	                    #sFB_Conveyor570(iUDT_ConveyorConfiguration := #iUDT_Configuration."570".Conveyor,
	                                     idi_PECEoSDistance := #iUDT_Configuration."570".PEC_Eos.Distance,
	                                     idi_PECBoSDistance := 0,
	                                     ii_ExternalSpeed := 0,
	                                     ix_SafetyOk := #ix_SafetyOk,
	                                     ix_24vOk := #ix_24vOk,
	                                     ix_400vOk := #ix_400vOk,
	                                     ix_HardwareOk := #iUDT_HardwareOk."570",
	                                     ix_PECEoS := #iqUDT_WorkstationStatus."570".PEC_EoS.PEC,
	                                     ix_PECBoS := TRUE,
	                                     ix_ExternalRequestHold := #sx_RightExternalRequestHold570,
	                                     qUDT_HMIStatus => #iqUDT_WorkstationStatus."570".Conveyor,
	                                     qUDT_Status => #iqUDT_WorkstationCommonStatus."570",
	                                     iqUDT_EquipmentControl := #iqUDT_EquipmentControl,
	                                     iqUDT_ConveyorCommand := #iqUDT_WorkstationCommands."570".Conveyor,
	                                     iqUDT_ConveyorInterface := #sUDT_Interface570,
	                                     iqUDT_HandShakeUp := #sUDT_Handshake560,
	                                     iqUDT_HandShake := #sUDT_Handshake570,
	                                     iqUDT_Statistics := #iqUDT_WorkstationStatistics."570".Conveyor);
	                END_REGION

	                REGION MCO

	                    #sFB_MCOConveyLinxAixController570(iUDT_AixConfig := #iUDT_Configuration."570".MCO_M01,
	                                                       iv_AixInputsModule := #iUDT_MotorInput570,
	                                                       ix_24vOk := #ix_24vOk,
	                                                       ix_SimulationModeActive := "DB_Memory".Simulation,
	                                                       ii_MotorPositionId := 1,
	                                                       qUDT_HMIStatus => #iqUDT_WorkstationStatus."570".MCO_M01,
	                                                       iqv_AixOutputsModule := #iqUDT_MotorOutput570,
	                                                       iqUDT_ConveyorInterface := #sUDT_Interface570,
	                                                       iqUDT_MCOStatistics := #iqUDT_WorkstationStatistics."570".MCO_M01);
	                END_REGION
	            END_REGION

	            REGION 580

	                REGION Displacement

	                    #sFB_Displacement580(#sUDT_Interface580);

	                END_REGION

	                REGION Tracking

	                    #sFB_Tracking580(iUDT_ConveyorCommonConfiguration := #iUDT_Configuration."580".Conveyor.Common,
	                                     iqa_TrackingData := #sa_TrackingArray580,
	                                     iqUDT_ConveyorInterface := #sUDT_Interface580,
	                                     iqUDT_HandshakeUp := #sUDT_Handshake570,
	                                     iqUDT_Handshake := #sUDT_Handshake580);
	                END_REGION

	                REGION EOS

	                    #sFB_PECUpdate580(iUDT_PECUpdateConfiguration := #iUDT_Configuration."580".PEC_Eos,
	                                      iUDT_ConveyorCommonConfiguration := #iUDT_Configuration."580".Conveyor.Common,
	                                      ix_PEC := NOT #iUDT_MotorInput570.AllSensorPortInputs.RightSensor,
	                                      ix_TeachingMode := FALSE,
	                                      qUDT_Status => #iqUDT_WorkstationStatus."580".PEC_EoS,
	                                      qi_GINwrite => #ti_dummy,
	                                      qx_PECFiltered => #tx_dummy,
	                                      iqa_TrackingData := #sa_TrackingArray580,
	                                      iqUDT_ConveyorInterface := #sUDT_Interface580,
	                                      iqUDT_UnknownGINRange := #iqUDT_UnknownGINRange,
	                                      iqUDT_FifoHeader := "DB_FIFOLostGIN".Header,
	                                      iqa_FifoData := "DB_FIFOLostGIN".Data,
	                                      iqUDT_Statistics := #iqUDT_WorkstationStatistics."580".PEC_EoS);

	                END_REGION

	                REGION Conveyor

	                    #sUDT_Handshake580.RTR := #sx_RightIndexing AND
	                    ((#iqUDT_WorkstationStatus."590".PEC_EoS.PEC AND #sUDT_Interface590.ActualSpeed <> 0) OR #iqUDT_WorkstationStatus."580".PEC_EoS.PEC);

	                    #sFB_Conveyor580(iUDT_ConveyorConfiguration := #iUDT_Configuration."580".Conveyor,
	                                     idi_PECEoSDistance := #iUDT_Configuration."580".PEC_Eos.Distance,
	                                     idi_PECBoSDistance := 0,
	                                     ii_ExternalSpeed := 0,
	                                     ix_SafetyOk := #ix_SafetyOk,
	                                     ix_24vOk := #ix_24vOk,
	                                     ix_400vOk := #ix_400vOk,
	                                     ix_HardwareOk := #iUDT_HardwareOk."580",
	                                     ix_PECEoS := #iqUDT_WorkstationStatus."580".PEC_EoS.PEC,
	                                     ix_PECBoS := TRUE,
	                                     ix_ReverseDirection := FALSE,
	                                     ix_ExternalRequestDieBack := FALSE,
	                                     ix_ExternalRequestHold := #sx_RightExternalRequestHold580,
	                                     ix_ResetEnergySave := FALSE,
	                                     qUDT_HMIStatus => #iqUDT_WorkstationStatus."580".Conveyor,
	                                     qUDT_Status => #iqUDT_WorkstationCommonStatus."580",
	                                     iqUDT_EquipmentControl := #iqUDT_EquipmentControl,
	                                     iqUDT_ConveyorCommand := #iqUDT_WorkstationCommands."580".Conveyor,
	                                     iqUDT_ConveyorInterface := #sUDT_Interface580,
	                                     iqUDT_HandShakeUp := #sUDT_Handshake570,
	                                     iqUDT_HandShake := #sUDT_Handshake580,
	                                     iqUDT_Statistics := #iqUDT_WorkstationStatistics."580".Conveyor);
	                END_REGION

	                REGION MCO

	                    #sFB_MCOConveyLinxAixController580(iUDT_AixConfig := #iUDT_Configuration."580".MCO_M01,
	                                                       iv_AixInputsModule := #iUDT_MotorInput570,
	                                                       ix_24vOk := #ix_24vOk,
	                                                       ix_SimulationModeActive := "DB_Memory".Simulation,
	                                                       ii_MotorPositionId := 2,
	                                                       qUDT_HMIStatus => #iqUDT_WorkstationStatus."580".MCO_M01,
	                                                       iqv_AixOutputsModule := #iqUDT_MotorOutput570,
	                                                       iqUDT_ConveyorInterface := #sUDT_Interface580,
	                                                       iqUDT_MCOStatistics := #iqUDT_WorkstationStatistics."580".MCO_M01);
	                END_REGION

	            END_REGION

	            REGION 590

	                REGION Displacement

	                    #sFB_Displacement590(#sUDT_Interface590);

	                END_REGION

	                REGION Tracking

	                    #sFB_Tracking590(iUDT_ConveyorCommonConfiguration := #iUDT_Configuration."590".Conveyor.Common,
	                                     iqa_TrackingData := #sa_TrackingArray590,
	                                     iqUDT_ConveyorInterface := #sUDT_Interface590,
	                                     iqUDT_HandshakeUp := #sUDT_Handshake580,
	                                     iqUDT_Handshake := #sUDT_Handshake590);
	                END_REGION

	                REGION EOS

	                    #sFB_PECUpdate590(iUDT_PECUpdateConfiguration := #iUDT_Configuration."590".PEC_Eos,
	                                      iUDT_ConveyorCommonConfiguration := #iUDT_Configuration."590".Conveyor.Common,
	                                      ix_PEC := NOT #iUDT_MotorInput590.AllSensorPortInputs.LeftSensor,
	                                      ix_TeachingMode := FALSE,
	                                      qUDT_Status => #iqUDT_WorkstationStatus."590".PEC_EoS,
	                                      qi_GINwrite => #ti_dummy,
	                                      qx_PECFiltered => #tx_dummy,
	                                      iqa_TrackingData := #sa_TrackingArray590,
	                                      iqUDT_ConveyorInterface := #sUDT_Interface590,
	                                      iqUDT_UnknownGINRange := #iqUDT_UnknownGINRange,
	                                      iqUDT_FifoHeader := "DB_FIFOLostGIN".Header,
	                                      iqa_FifoData := "DB_FIFOLostGIN".Data,
	                                      iqUDT_Statistics := #iqUDT_WorkstationStatistics."590".PEC_EoS);

	                END_REGION

	                REGION Conveyor

	                    #sUDT_Handshake590.RTR := (#sx_RightIndexing AND #iqUDT_WorkstationStatus."590".PEC_EoS.PEC)
	                    OR (#sx_RightPushOutActiveStation1 AND #iqUDT_WorkstationStatus."610".PEC_EoS.PEC AND #sUDT_Interface611.ActualSpeed <> 0);

	                    #sFB_Conveyor590(iUDT_ConveyorConfiguration := #iUDT_Configuration."590".Conveyor,
	                                     idi_PECEoSDistance := #iUDT_Configuration."590".PEC_Eos.Distance,
	                                     idi_PECBoSDistance := 0,
	                                     ii_ExternalSpeed := 0,
	                                     ix_SafetyOk := #ix_SafetyOk,
	                                     ix_24vOk := #ix_24vOk,
	                                     ix_400vOk := #ix_400vOk,
	                                     ix_HardwareOk := #iUDT_HardwareOk."590",
	                                     ix_PECEoS := #iqUDT_WorkstationStatus."590".PEC_EoS.PEC,
	                                     ix_PECBoS := TRUE,
	                                     ix_ReverseDirection := FALSE,
	                                     ix_ExternalRequestDieBack := FALSE,
	                                     ix_ExternalRequestHold := #sx_RightExternalRequestHold590,
	                                     ix_ResetEnergySave := FALSE,
	                                     qUDT_HMIStatus => #iqUDT_WorkstationStatus."590".Conveyor,
	                                     qUDT_Status => #iqUDT_WorkstationCommonStatus."590",
	                                     iqUDT_EquipmentControl := #iqUDT_EquipmentControl,
	                                     iqUDT_ConveyorCommand := #iqUDT_WorkstationCommands."590".Conveyor,
	                                     iqUDT_ConveyorInterface := #sUDT_Interface590,
	                                     iqUDT_HandShakeUp := #sUDT_Handshake580,
	                                     iqUDT_HandShake := #sUDT_Handshake590,
	                                     iqUDT_Statistics := #iqUDT_WorkstationStatistics."590".Conveyor);
	                END_REGION

	                REGION MCO

	                    #sFB_MCOConveyLinxAixController590(iUDT_AixConfig := #iUDT_Configuration."590".MCO_M01,
	                                                       iv_AixInputsModule := #iUDT_MotorInput590,
	                                                       ix_24vOk := #ix_24vOk,
	                                                       ix_SimulationModeActive := "DB_Memory".Simulation,
	                                                       ii_MotorPositionId := 1,
	                                                       qUDT_HMIStatus => #iqUDT_WorkstationStatus."590".MCO_M01,
	                                                       iqv_AixOutputsModule := #iqUDT_MotorOutput590,
	                                                       iqUDT_ConveyorInterface := #sUDT_Interface590,
	                                                       iqUDT_MCOStatistics := #iqUDT_WorkstationStatistics."590".MCO_M01);
	                END_REGION
	            END_REGION

	            REGION 610

	                REGION Displacement

	                    #sFB_Displacement610(#sUDT_Interface610);

	                END_REGION

	                REGION MCO

	                    #sFB_MCOConveyLinxAixController610(iUDT_AixConfig := #iUDT_Configuration."610".MCO_M01,
	                                                       iv_AixInputsModule := #iUDT_MotorInput610,
	                                                       ix_24vOk := #ix_24vOk,
	                                                       ix_SimulationModeActive := "DB_Memory".Simulation,
	                                                       ii_MotorPositionId := 1,
	                                                       qUDT_HMIStatus => #iqUDT_WorkstationStatus."610".MCO_M01,
	                                                       iqv_AixOutputsModule := #iqUDT_MotorOutput610,
	                                                       iqUDT_ConveyorInterface := #sUDT_Interface610,
	                                                       iqUDT_MCOStatistics := #iqUDT_WorkstationStatistics."610".MCO_M01);
	                END_REGION
	            END_REGION

	            REGION 611

	                REGION Displacement

	                    #sFB_Displacement611(#sUDT_Interface611);

	                END_REGION

	                REGION RAT

	                    #sFB_RightAngledTransfer611(iUDT_Configuration := #iUDT_Configuration."611".RightAngledTransfer,
	                                                iUDT_LowerConveyorConfiguration := #iUDT_Configuration."610".Conveyor,
	                                                iUDT_UpperConveyorConfiguration := #iUDT_Configuration."611".Conveyor,
	                                                iUDT_PECConfiguration := #iUDT_Configuration."610".PEC_EoS,
	                                                ii_DestinationA := 0,
	                                                ii_DestinationB := 0,
	                                                ii_DestinationC := 0,
	                                                ii_DestinationD := 2,
	                                                ix_HardwareOk := #iUDT_HardwareOk."610",
	                                                ix_400vOk := #ix_400vOk,
	                                                ix_24vOk := #ix_24vOk,
	                                                ix_SafetyOk := #ix_SafetyOk,
	                                                ix_AirPressureOk := #ix_AirPressureOk,
	                                                ix_SectionIsDown := #ix_SectionIsDown611,
	                                                ix_SectionIsUp := #ix_SectionIsUp611,
	                                                ix_ConveyorAAuto := false,
	                                                ix_ConveyorBAuto := false,
	                                                ix_ConveyorCAuto := FALSE,
	                                                ix_ConveyorDAuto := #iqUDT_WorkstationCommonStatus."590".AutoON,
	                                                ix_PEC := #iUDT_MotorInput610.AllSensorPortInputs.LeftSensor,
	                                                ix_ExternalReceiveRequestA := FALSE,
	                                                ix_ExternalReceiveRequestB := FALSE,
	                                                ix_ExternalReceiveRequestC := FALSE,
	                                                ix_ExternalReceiveRequestD := #sx_RightPushOutActiveStation1,
	                                                ix_PECInfeedD := #iqUDT_WorkstationStatus."590".PEC_EoS.PEC,
	                                                qUDT_HMIRATStatus => #iqUDT_WorkstationStatus."611".RightAngledTransfer,
	                                                qUDT_HMIConveyorStatus => #iqUDT_WorkstationStatus."610".Conveyor,
	                                                qUDT_HMIPECStatus => #iqUDT_WorkstationStatus."610".PEC_EoS,
	                                                qUDT_RATStatus => #iqUDT_WorkstationCommonStatus."611",
	                                                qUDT_ConveyorStatus => #iqUDT_WorkstationCommonStatus."610",
	                                                qx_PopupControl => #qx_PopupControl611,
	                                                qx_ExternalSendRequestA => #tx_dummy,
	                                                qx_ExternalSendRequestB => #tx_dummy,
	                                                qx_ExternalSendRequestC => #tx_dummy,
	                                                qx_ExternalSendRequestD => #tx_dummy,
	                                                iqUDT_EquipmentControl := #iqUDT_EquipmentControl,
	                                                iqUDT_RATCommand := #iqUDT_WorkstationCommands."611".RightAngledTransfer,
	                                                iqUDT_ConveyorCommand := #iqUDT_WorkstationCommands."610".Conveyor,
	                                                iqUDT_RATStatistics := #iqUDT_WorkstationStatistics."611".RightAngledTransfer,
	                                                iqUDT_ConveyorStatistics := #iqUDT_WorkstationStatistics."610".Conveyor,
	                                                iqUDT_PECStatistics := #iqUDT_WorkstationStatistics."610".PEC_EoS,
	                                                iqUDT_HandShakeConveyorA := #tUDT_DummyConveyorHandshake,
	                                                iqUDT_HandShakeConveyorB := #sUDT_Handshake610,
	                                                iqUDT_HandShakeConveyorC := #sUDT_Handshake590,
	                                                iqUDT_HandShakeConveyorD := #tUDT_DummyConveyorHandshake,
	                                                iqUDT_LowerConveyorInterface := #sUDT_Interface610,
	                                                iqUDT_UpperConveyorInterface := #sUDT_Interface611,
	                                                iqUDT_RATPositioning := #iqUDT_RATPositioning610,
	                                                iqUDT_BladeStopEoSInterface := #tUDT_DummyBladeStop,
	                                                iqUDT_BladeStopBoSInterface := #tUDT_DummyBladeStop);

	                END_REGION

	                REGION MCO

	                    #sFB_MCOConveyLinxAixController611(iUDT_AixConfig := #iUDT_Configuration."611".MCO_M01,
	                                                       iv_AixInputsModule := #iUDT_MotorInput610,
	                                                       ii_PositionSetpoint := #iqUDT_RATPositioning610.Upper.EndPosition,
	                                                       ix_24vOk := #ix_24vOk,
	                                                       ix_SimulationModeActive := "DB_Memory".Simulation,
	                                                       ii_MotorPositionId := 2,
	                                                       ix_StartPositioning := #iqUDT_RATPositioning610.Upper.Start,
	                                                       ix_ResetPosition := #iqUDT_RATPositioning610.Upper.ResetPosition,
	                                                       qUDT_HMIStatus => #iqUDT_WorkstationStatus."611".MCO_M01,
	                                                       qx_Positioned => #iqUDT_RATPositioning610.Upper.Done,
	                                                       iqv_AixOutputsModule := #iqUDT_MotorOutput610,
	                                                       iqUDT_ConveyorInterface := #sUDT_Interface611,
	                                                       iqUDT_MCOStatistics := #iqUDT_WorkstationStatistics."611".MCO_M01);
	                END_REGION

	            END_REGION

	            REGION 620

	                REGION Displacement

	                    #sFB_Displacement620(#sUDT_Interface620);

	                END_REGION

	                REGION MCO

	                    #sFB_MCOConveyLinxAixController620(iUDT_AixConfig := #iUDT_Configuration."620".MCO_M01,
	                                                       iv_AixInputsModule := #iUDT_MotorInput620,
	                                                       ii_PositionSetpoint := #iqUDT_RATPositioning620.Lower.EndPosition,
	                                                       ix_24vOk := #ix_24vOk,
	                                                       ix_SimulationModeActive := "DB_Memory".Simulation,
	                                                       ii_MotorPositionId := 1,
	                                                       ix_StartPositioning := #iqUDT_RATPositioning620.Lower.Start,
	                                                       ix_ResetPosition := #iqUDT_RATPositioning620.Lower.ResetPosition,
	                                                       qUDT_HMIStatus => #iqUDT_WorkstationStatus."620".MCO_M01,
	                                                       qx_Positioned => #iqUDT_RATPositioning620.Lower.Done,
	                                                       iqv_AixOutputsModule := #iqUDT_MotorOutput620,
	                                                       iqUDT_ConveyorInterface := #sUDT_Interface620,
	                                                       iqUDT_MCOStatistics := #iqUDT_WorkstationStatistics."620".MCO_M01);
	                END_REGION
	            END_REGION

	            REGION 621

	                REGION Displacement

	                    #sFB_Displacement621(#sUDT_Interface621);

	                END_REGION

	                REGION RAT

	                    #sFB_RightAngledTransfer621(iUDT_Configuration := #iUDT_Configuration."621".RightAngledTransfer,
	                                                iUDT_LowerConveyorConfiguration := #iUDT_Configuration."620".Conveyor,
	                                                iUDT_UpperConveyorConfiguration := #iUDT_Configuration."621".Conveyor,
	                                                iUDT_PECConfiguration := #iUDT_Configuration."620".PEC_EoS,
	                                                ii_DestinationA := 2,
	                                                ii_DestinationB := 0,
	                                                ii_DestinationC := 0,
	                                                ii_DestinationD := 2,
	                                                ix_HardwareOk := #iUDT_HardwareOk."620",
	                                                ix_400vOk := #ix_400vOk,
	                                                ix_24vOk := #ix_24vOk,
	                                                ix_SafetyOk := #ix_SafetyOk,
	                                                ix_AirPressureOk := #ix_AirPressureOk,
	                                                ix_SectionIsDown := #ix_SectionIsDown621,
	                                                ix_SectionIsUp := #ix_SectionIsUp621,
	                                                ix_ConveyorAAuto := #iqUDT_WorkstationCommonStatus."610".AutoON,
	                                                ix_ConveyorBAuto := false,
	                                                ix_ConveyorCAuto := false,
	                                                ix_ConveyorDAuto := #iqUDT_WorkstationCommonStatus."750".AutoON,
	                                                ix_PEC := #iUDT_MotorInput620.AllSensorPortInputs.LeftSensor,
	                                                ix_ExternalReceiveRequestA := NOT #iqUDT_WorkstationStatus."610".PEC_EoS.PEC,
	                                                ix_ExternalReceiveRequestB := FALSE,
	                                                ix_ExternalReceiveRequestC := FALSE,
	                                                ix_ExternalReceiveRequestD := NOT #iqUDT_WorkstationStatus."750".PEC_EoS.PEC,
	                                                ix_PECInfeedA := #iqUDT_WorkstationStatus."610".PEC_EoS.PEC,
	                                                ix_PECInfeedD := #iqUDT_WorkstationStatus."750".PEC_EoS.PEC,
	                                                qUDT_HMIRATStatus => #iqUDT_WorkstationStatus."621".RightAngledTransfer,
	                                                qUDT_HMIConveyorStatus => #iqUDT_WorkstationStatus."620".Conveyor,
	                                                qUDT_HMIPECStatus => #iqUDT_WorkstationStatus."620".PEC_EoS,
	                                                qUDT_RATStatus => #iqUDT_WorkstationCommonStatus."621",
	                                                qUDT_ConveyorStatus => #iqUDT_WorkstationCommonStatus."620",
	                                                qx_PopupControl => #qx_PopupControl621,
	                                                qx_ExternalSendRequestA => #tx_dummy,
	                                                qx_ExternalSendRequestB => #tx_dummy,
	                                                qx_ExternalSendRequestC => #tx_dummy,
	                                                qx_ExternalSendRequestD => #tx_dummy,
	                                                iqUDT_EquipmentControl := #iqUDT_EquipmentControl,
	                                                iqUDT_RATCommand := #iqUDT_WorkstationCommands."621".RightAngledTransfer,
	                                                iqUDT_ConveyorCommand := #iqUDT_WorkstationCommands."620".Conveyor,
	                                                iqUDT_RATStatistics := #iqUDT_WorkstationStatistics."621".RightAngledTransfer,
	                                                iqUDT_ConveyorStatistics := #iqUDT_WorkstationStatistics."620".Conveyor,
	                                                iqUDT_PECStatistics := #iqUDT_WorkstationStatistics."620".PEC_EoS,
	                                                iqUDT_HandShakeConveyorA := #sUDT_Handshake610,
	                                                iqUDT_HandShakeConveyorB := #iqUDT_HandshakeDownstream620,
	                                                iqUDT_HandShakeConveyorC := #tUDT_DummyConveyorHandshake,
	                                                iqUDT_HandShakeConveyorD := #sUDT_Handshake750,
	                                                iqUDT_LowerConveyorInterface := #sUDT_Interface620,
	                                                iqUDT_UpperConveyorInterface := #sUDT_Interface621,
	                                                iqUDT_RATPositioning := #iqUDT_RATPositioning620,
	                                                iqUDT_BladeStopEoSInterface := #tUDT_DummyBladeStop,
	                                                iqUDT_BladeStopBoSInterface := #tUDT_DummyBladeStop);

	                END_REGION

	                REGION MCO

	                    #sFB_MCOConveyLinxAixController621(iUDT_AixConfig := #iUDT_Configuration."621".MCO_M01,
	                                                       iv_AixInputsModule := #iUDT_MotorInput620,
	                                                       ii_PositionSetpoint := #iqUDT_RATPositioning620.Upper.EndPosition,
	                                                       ix_24vOk := #ix_24vOk,
	                                                       ix_SimulationModeActive := "DB_Memory".Simulation,
	                                                       ii_MotorPositionId := 2,
	                                                       ix_StartPositioning := #iqUDT_RATPositioning620.Upper.Start,
	                                                       ix_ResetPosition := #iqUDT_RATPositioning620.Upper.ResetPosition,
	                                                       qUDT_HMIStatus => #iqUDT_WorkstationStatus."621".MCO_M01,
	                                                       qx_Positioned => #iqUDT_RATPositioning620.Upper.Done,
	                                                       iqv_AixOutputsModule := #iqUDT_MotorOutput620,
	                                                       iqUDT_ConveyorInterface := #sUDT_Interface621,
	                                                       iqUDT_MCOStatistics := #iqUDT_WorkstationStatistics."621".MCO_M01);
	                END_REGION

	            END_REGION

	            REGION 710

	                REGION Displacement

	                    #sFB_Displacement710(#sUDT_Interface710);

	                END_REGION

	                REGION EOS
	                    #sFB_PEC710(ix_PEC := NOT #iUDT_MotorInput710.AllSensorPortInputs.LeftSensor,
	                                iUDT_PECConfiguration := #iUDT_Configuration."710".PEC_Eos,
	                                qx_PECFiltered => #tx_dummy,
	                                qUDT_HMIStatus => #iqUDT_WorkstationStatus."710".PEC_EoS,
	                                iqUDT_ConveyorInterface := #sUDT_Interface710,
	                                iqUDT_PECStatistics := #iqUDT_WorkstationStatistics."710".PEC_EoS);

	                END_REGION

	                REGION Conveyor

	                    #sFB_Conveyor710(iUDT_ConveyorConfiguration := #iUDT_Configuration."710".Conveyor,
	                                     idi_PECEoSDistance := #iUDT_Configuration."710".PEC_Eos.Distance,
	                                     idi_PECBoSDistance := 0,
	                                     ii_ExternalSpeed := 0,
	                                     ix_SafetyOk := #ix_SafetyOk,
	                                     ix_24vOk := #ix_24vOk,
	                                     ix_400vOk := #ix_400vOk,
	                                     ix_HardwareOk := #iUDT_HardwareOk."710",
	                                     ix_PECEoS := #iqUDT_WorkstationStatus."710".PEC_EoS.PEC,
	                                     ix_PECBoS := TRUE,
	                                     ix_ReverseDirection := FALSE,
	                                     ix_ExternalRequestDieBack := FALSE,
	                                     ix_ExternalRequestHold := #sx_RightExternalRequestHold710,
	                                     ix_ResetEnergySave := FALSE,
	                                     qUDT_HMIStatus => #iqUDT_WorkstationStatus."710".Conveyor,
	                                     qUDT_Status => #iqUDT_WorkstationCommonStatus."710",
	                                     iqUDT_EquipmentControl := #iqUDT_EquipmentControl,
	                                     iqUDT_ConveyorCommand := #iqUDT_WorkstationCommands."710".Conveyor,
	                                     iqUDT_ConveyorInterface := #sUDT_Interface710,
	                                     iqUDT_HandShakeUp := #tUDT_DummyConveyorHandshake,
	                                     iqUDT_HandShake := #sUDT_Handshake710,
	                                     iqUDT_Statistics := #iqUDT_WorkstationStatistics."710".Conveyor);
	                END_REGION

	                REGION MCO

	                    #sFB_MCOConveyLinxAixController710(iUDT_AixConfig := #iUDT_Configuration."710".MCO_M01,
	                                                       iv_AixInputsModule := #iUDT_MotorInput710,
	                                                       ix_24vOk := #ix_24vOk,
	                                                       ix_SimulationModeActive := "DB_Memory".Simulation,
	                                                       ii_MotorPositionId := 1,
	                                                       qUDT_HMIStatus => #iqUDT_WorkstationStatus."710".MCO_M01,
	                                                       iqv_AixOutputsModule := #iqUDT_MotorOutput710,
	                                                       iqUDT_ConveyorInterface := #sUDT_Interface710,
	                                                       iqUDT_MCOStatistics := #iqUDT_WorkstationStatistics."710".MCO_M01);
	                END_REGION

	            END_REGION

	            REGION 720

	                REGION Displacement

	                    #sFB_Displacement720(#sUDT_Interface720);

	                END_REGION

	                REGION EOS
	                    #sFB_PEC720(ix_PEC := NOT #iUDT_MotorInput710.AllSensorPortInputs.RightSensor,
	                                iUDT_PECConfiguration := #iUDT_Configuration."720".PEC_Eos,
	                                qx_PECFiltered => #tx_dummy,
	                                qUDT_HMIStatus => #iqUDT_WorkstationStatus."720".PEC_EoS,
	                                iqUDT_ConveyorInterface := #sUDT_Interface720,
	                                iqUDT_PECStatistics := #iqUDT_WorkstationStatistics."720".PEC_EoS);


	                END_REGION

	                REGION Conveyor

	                    #sFB_Conveyor720(iUDT_ConveyorConfiguration := #iUDT_Configuration."720".Conveyor,
	                                     idi_PECEoSDistance := #iUDT_Configuration."720".PEC_Eos.Distance,
	                                     idi_PECBoSDistance := 0,
	                                     ii_ExternalSpeed := 0,
	                                     ix_SafetyOk := #ix_SafetyOk,
	                                     ix_24vOk := #ix_24vOk,
	                                     ix_400vOk := #ix_400vOk,
	                                     ix_HardwareOk := #iUDT_HardwareOk."710",
	                                     ix_PECEoS := #iqUDT_WorkstationStatus."720".PEC_EoS.PEC,
	                                     ix_PECBoS := TRUE,
	                                     ix_ReverseDirection := FALSE,
	                                     ix_ExternalRequestDieBack := FALSE,
	                                     ix_ExternalRequestHold := #sx_RightExternalRequestHold720,
	                                     ix_ResetEnergySave := FALSE,
	                                     qUDT_HMIStatus => #iqUDT_WorkstationStatus."720".Conveyor,
	                                     qUDT_Status => #iqUDT_WorkstationCommonStatus."720",
	                                     iqUDT_EquipmentControl := #iqUDT_EquipmentControl,
	                                     iqUDT_ConveyorCommand := #iqUDT_WorkstationCommands."720".Conveyor,
	                                     iqUDT_ConveyorInterface := #sUDT_Interface720,
	                                     iqUDT_HandShakeUp := #sUDT_Handshake710,
	                                     iqUDT_HandShake := #sUDT_Handshake720,
	                                     iqUDT_Statistics := #iqUDT_WorkstationStatistics."720".Conveyor);
	                END_REGION

	                REGION MCO

	                    #sFB_MCOConveyLinxAixController720(iUDT_AixConfig := #iUDT_Configuration."720".MCO_M01,
	                                                       iv_AixInputsModule := #iUDT_MotorInput710,
	                                                       ix_24vOk := #ix_24vOk,
	                                                       ix_SimulationModeActive := "DB_Memory".Simulation,
	                                                       ii_MotorPositionId := 2,
	                                                       qUDT_HMIStatus => #iqUDT_WorkstationStatus."720".MCO_M01,
	                                                       iqv_AixOutputsModule := #iqUDT_MotorOutput710,
	                                                       iqUDT_ConveyorInterface := #sUDT_Interface720,
	                                                       iqUDT_MCOStatistics := #iqUDT_WorkstationStatistics."720".MCO_M01);
	                END_REGION

	            END_REGION

	            REGION 730

	                REGION Displacement

	                    #sFB_Displacement730(#sUDT_Interface730);

	                END_REGION

	                REGION EOS
	                    #sFB_PEC730(ix_PEC := NOT #iUDT_MotorInput730.AllSensorPortInputs.LeftSensor,
	                                iUDT_PECConfiguration := #iUDT_Configuration."730".PEC_Eos,
	                                qx_PECFiltered => #tx_dummy,
	                                qUDT_HMIStatus => #iqUDT_WorkstationStatus."730".PEC_EoS,
	                                iqUDT_ConveyorInterface := #sUDT_Interface730,
	                                iqUDT_PECStatistics := #iqUDT_WorkstationStatistics."730".PEC_EoS);


	                END_REGION

	                REGION Conveyor

	                    #sFB_Conveyor730(iUDT_ConveyorConfiguration := #iUDT_Configuration."730".Conveyor,
	                                     idi_PECEoSDistance := #iUDT_Configuration."730".PEC_Eos.Distance,
	                                     idi_PECBoSDistance := 0,
	                                     ii_ExternalSpeed := 0,
	                                     ix_SafetyOk := #ix_SafetyOk,
	                                     ix_24vOk := #ix_24vOk,
	                                     ix_400vOk := #ix_400vOk,
	                                     ix_HardwareOk := #iUDT_HardwareOk."730",
	                                     ix_PECEoS := #iqUDT_WorkstationStatus."730".PEC_EoS.PEC,
	                                     ix_PECBoS := TRUE,
	                                     ix_ReverseDirection := FALSE,
	                                     ix_ExternalRequestDieBack := FALSE,
	                                     ix_ExternalRequestHold := #sx_RightExternalRequestHold730,
	                                     ix_ResetEnergySave := FALSE,
	                                     qUDT_HMIStatus => #iqUDT_WorkstationStatus."730".Conveyor,
	                                     qUDT_Status => #iqUDT_WorkstationCommonStatus."730",
	                                     iqUDT_EquipmentControl := #iqUDT_EquipmentControl,
	                                     iqUDT_ConveyorCommand := #iqUDT_WorkstationCommands."730".Conveyor,
	                                     iqUDT_ConveyorInterface := #sUDT_Interface730,
	                                     iqUDT_HandShakeUp := #sUDT_Handshake720,
	                                     iqUDT_HandShake := #sUDT_Handshake730,
	                                     iqUDT_Statistics := #iqUDT_WorkstationStatistics."730".Conveyor);
	                END_REGION

	                REGION MCO

	                    #sFB_MCOConveyLinxAixController730(iUDT_AixConfig := #iUDT_Configuration."730".MCO_M01,
	                                                       iv_AixInputsModule := #iUDT_MotorInput730,
	                                                       ix_24vOk := #ix_24vOk,
	                                                       ix_SimulationModeActive := "DB_Memory".Simulation,
	                                                       ii_MotorPositionId := 1,
	                                                       qUDT_HMIStatus => #iqUDT_WorkstationStatus."730".MCO_M01,
	                                                       iqv_AixOutputsModule := #iqUDT_MotorOutput730,
	                                                       iqUDT_ConveyorInterface := #sUDT_Interface730,
	                                                       iqUDT_MCOStatistics := #iqUDT_WorkstationStatistics."730".MCO_M01);
	                END_REGION
	            END_REGION

	            REGION 740

	                REGION Displacement

	                    #sFB_Displacement740(#sUDT_Interface740);

	                END_REGION

	                REGION EOS
	                    #sFB_PEC740(ix_PEC := NOT #iUDT_MotorInput730.AllSensorPortInputs.RightSensor,
	                                iUDT_PECConfiguration := #iUDT_Configuration."740".PEC_Eos,
	                                qx_PECFiltered => #tx_dummy,
	                                qUDT_HMIStatus => #iqUDT_WorkstationStatus."740".PEC_EoS,
	                                iqUDT_ConveyorInterface := #sUDT_Interface740,
	                                iqUDT_PECStatistics := #iqUDT_WorkstationStatistics."740".PEC_EoS);


	                END_REGION


	                REGION Conveyor

	                    #sFB_Conveyor740(iUDT_ConveyorConfiguration := #iUDT_Configuration."740".Conveyor,
	                                     idi_PECEoSDistance := #iUDT_Configuration."740".PEC_Eos.Distance,
	                                     idi_PECBoSDistance := 0,
	                                     ii_ExternalSpeed := 0,
	                                     ix_SafetyOk := #ix_SafetyOk,
	                                     ix_24vOk := #ix_24vOk,
	                                     ix_400vOk := #ix_400vOk,
	                                     ix_HardwareOk := #iUDT_HardwareOk."730",
	                                     ix_PECEoS := #iqUDT_WorkstationStatus."740".PEC_EoS.PEC,
	                                     ix_PECBoS := TRUE,
	                                     ix_ReverseDirection := FALSE,
	                                     ix_ExternalRequestDieBack := FALSE,
	                                     ix_ExternalRequestHold := #sx_RightExternalRequestHold740,
	                                     ix_ResetEnergySave := FALSE,
	                                     qUDT_HMIStatus => #iqUDT_WorkstationStatus."740".Conveyor,
	                                     qUDT_Status => #iqUDT_WorkstationCommonStatus."740",
	                                     iqUDT_EquipmentControl := #iqUDT_EquipmentControl,
	                                     iqUDT_ConveyorCommand := #iqUDT_WorkstationCommands."740".Conveyor,
	                                     iqUDT_ConveyorInterface := #sUDT_Interface740,
	                                     iqUDT_HandShakeUp := #sUDT_Handshake730,
	                                     iqUDT_HandShake := #sUDT_Handshake740,
	                                     iqUDT_Statistics := #iqUDT_WorkstationStatistics."740".Conveyor);
	                END_REGION

	                REGION MCO

	                    #sFB_MCOConveyLinxAixController740(iUDT_AixConfig := #iUDT_Configuration."740".MCO_M01,
	                                                       iv_AixInputsModule := #iUDT_MotorInput730,
	                                                       ix_24vOk := #ix_24vOk,
	                                                       ix_SimulationModeActive := "DB_Memory".Simulation,
	                                                       ii_MotorPositionId := 2,
	                                                       qUDT_HMIStatus => #iqUDT_WorkstationStatus."740".MCO_M01,
	                                                       iqv_AixOutputsModule := #iqUDT_MotorOutput730,
	                                                       iqUDT_ConveyorInterface := #sUDT_Interface740,
	                                                       iqUDT_MCOStatistics := #iqUDT_WorkstationStatistics."740".MCO_M01);
	                END_REGION

	            END_REGION

	            REGION 750

	                REGION Displacement

	                    #sFB_Displacement750(#sUDT_Interface750);

	                END_REGION

	                REGION EOS
	                    #sFB_PEC750(ix_PEC := NOT #iUDT_MotorInput750.AllSensorPortInputs.LeftSensor,
	                                iUDT_PECConfiguration := #iUDT_Configuration."750".PEC_Eos,
	                                qx_PECFiltered => #tx_dummy,
	                                qUDT_HMIStatus => #iqUDT_WorkstationStatus."750".PEC_EoS,
	                                iqUDT_ConveyorInterface := #sUDT_Interface750,
	                                iqUDT_PECStatistics := #iqUDT_WorkstationStatistics."750".PEC_EoS);

	                END_REGION

	                REGION Conveyor

	                    #sUDT_Handshake750.RTR := #sUDT_Handshake750.RTR OR #iqUDT_WorkstationStatus."750".PEC_EoS.PEC;

	                    #sFB_Conveyor750(iUDT_ConveyorConfiguration := #iUDT_Configuration."750".Conveyor,
	                                     idi_PECEoSDistance := #iUDT_Configuration."750".PEC_Eos.Distance,
	                                     idi_PECBoSDistance := 0,
	                                     ii_ExternalSpeed := 0,
	                                     ix_SafetyOk := #ix_SafetyOk,
	                                     ix_24vOk := #ix_24vOk,
	                                     ix_400vOk := #ix_400vOk,
	                                     ix_HardwareOk := #iUDT_HardwareOk."750",
	                                     ix_PECEoS := #iqUDT_WorkstationStatus."750".PEC_EoS.PEC,
	                                     ix_PECBoS := TRUE,
	                                     ix_ReverseDirection := FALSE,
	                                     ix_ExternalRequestDieBack := FALSE,
	                                     ix_ExternalRequestHold := #sx_RightExternalRequestHold750,
	                                     ix_ResetEnergySave := FALSE,
	                                     qUDT_HMIStatus => #iqUDT_WorkstationStatus."750".Conveyor,
	                                     qUDT_Status => #iqUDT_WorkstationCommonStatus."750",
	                                     iqUDT_EquipmentControl := #iqUDT_EquipmentControl,
	                                     iqUDT_ConveyorCommand := #iqUDT_WorkstationCommands."750".Conveyor,
	                                     iqUDT_ConveyorInterface := #sUDT_Interface750,
	                                     iqUDT_HandShakeUp := #sUDT_Handshake740,
	                                     iqUDT_HandShake := #sUDT_Handshake750,
	                                     iqUDT_Statistics := #iqUDT_WorkstationStatistics."750".Conveyor);
	                END_REGION

	                REGION MCO

	                    #sFB_MCOConveyLinxAixController750(iUDT_AixConfig := #iUDT_Configuration."750".MCO_M01,
	                                                       iv_AixInputsModule := #iUDT_MotorInput750,
	                                                       ix_24vOk := #ix_24vOk,
	                                                       ix_SimulationModeActive := "DB_Memory".Simulation,
	                                                       ii_MotorPositionId := 1,
	                                                       qUDT_HMIStatus => #iqUDT_WorkstationStatus."750".MCO_M01,
	                                                       iqv_AixOutputsModule := #iqUDT_MotorOutput750,
	                                                       iqUDT_ConveyorInterface := #sUDT_Interface750,
	                                                       iqUDT_MCOStatistics := #iqUDT_WorkstationStatistics."750".MCO_M01);
	                END_REGION
	            END_REGION

	            REGION 760
	                REGION Displacement
	                    #sFB_Displacement760(#sUDT_Interface760);

	                END_REGION


	                REGION Conveyor

	                    #sUDT_Handshake760.RTR := TRUE;

	                    #sFB_Conveyor760(iUDT_ConveyorConfiguration := #iUDT_Configuration."760".Conveyor,
	                                     ix_SafetyOk := #ix_SafetyOk,
	                                     ix_24vOk := #ix_24vOk,
	                                     ix_400vOk := #ix_400vOk,
	                                     ix_HardwareOk := #iUDT_HardwareOk."760",
	                                     ix_ExternalRequestHold := #sx_Hold760,
	                                     qUDT_HMIStatus => #iqUDT_WorkstationStatus."760".Conveyor,
	                                     qUDT_Status => #iqUDT_WorkstationCommonStatus."760",
	                                     iqUDT_EquipmentControl := #iqUDT_EquipmentControl,
	                                     iqUDT_ConveyorCommand := #iqUDT_WorkstationCommands."760".Conveyor,
	                                     iqUDT_ConveyorInterface := #sUDT_Interface760,
	                                     iqUDT_HandShakeUp := #sUDT_HandshakeUp760,
	                                     iqUDT_HandShake := #sUDT_Handshake760,
	                                     iqUDT_Statistics := #iqUDT_WorkstationStatistics."760".Conveyor);

	                END_REGION


	                REGION MCO

	                    #sFB_MCOConveyLinxAixController760(iUDT_AixConfig := #iUDT_Configuration."760".MCO_M01,
	                                                       iv_AixInputsModule := #iUDT_MotorInput760,
	                                                       ii_MotorPositionId := 1,
	                                                       ix_24vOk := #ix_24vOk,
	                                                       ix_SimulationModeActive := "DB_Memory".Simulation,
	                                                       qUDT_HMIStatus => #iqUDT_WorkstationStatus."760".MCO_M01,
	                                                       iqv_AixOutputsModule := #iqUDT_MotorOutput760,
	                                                       iqUDT_ConveyorInterface := #sUDT_Interface760,
	                                                       iqUDT_MCOStatistics := #iqUDT_WorkstationStatistics."760".MCO_M01);
	                END_REGION

	            END_REGION

	            REGION 770

	                REGION Displacement
	                    #sFB_Displacement760(#sUDT_Interface770);
	                END_REGION

	                REGION Conveyor

	                    #sUDT_Handshake770.RTR := TRUE;

	                    #sFB_Conveyor770(iUDT_ConveyorConfiguration := #iUDT_Configuration."770".Conveyor,
	                                     ix_SafetyOk := #ix_SafetyOk,
	                                     ix_24vOk := #ix_24vOk,
	                                     ix_400vOk := #ix_400vOk,
	                                     ix_HardwareOk := #iUDT_HardwareOk."760",
	                                     ix_ExternalRequestHold := #sx_Hold770,
	                                     qUDT_HMIStatus => #iqUDT_WorkstationStatus."770".Conveyor,
	                                     qUDT_Status => #iqUDT_WorkstationCommonStatus."770",
	                                     iqUDT_EquipmentControl := #iqUDT_EquipmentControl,
	                                     iqUDT_ConveyorCommand := #iqUDT_WorkstationCommands."770".Conveyor,
	                                     iqUDT_ConveyorInterface := #sUDT_Interface770,
	                                     iqUDT_HandShakeUp := #sUDT_HandshakeUp770,
	                                     iqUDT_HandShake := #sUDT_Handshake770,
	                                     iqUDT_Statistics := #iqUDT_WorkstationStatistics."770".Conveyor);

	                END_REGION

	                REGION MCO
	                    #sFB_MCOConveyLinxAixController770(iUDT_AixConfig := #iUDT_Configuration."770".MCO_M01,
	                                                       iv_AixInputsModule := #iUDT_MotorInput760,
	                                                       ii_MotorPositionId := 2,
	                                                       ix_24vOk := #ix_24vOk,
	                                                       ix_SimulationModeActive := "DB_Memory".Simulation,
	                                                       qUDT_HMIStatus => #iqUDT_WorkstationStatus."770".MCO_M01,
	                                                       iqv_AixOutputsModule := #iqUDT_MotorOutput760,
	                                                       iqUDT_ConveyorInterface := #sUDT_Interface770,
	                                                       iqUDT_MCOStatistics := #iqUDT_WorkstationStatistics."770".MCO_M01);
	                END_REGION
	            END_REGION
	        END_REGION

	    END_IF;

	END_REGION

	IF #iUDT_Configuration.GlobalConfig.StationVariant = 3 THEN

	    #iqUDT_RightWESInterface := #iqUDT_LeftWESInterface;

	END_IF;


END_FUNCTION_BLOCK

